TYPE XtsPartStatus :
STRUCT
	PartDriveState: Tc3_XTS_Utility.DriveState;
	IsDCLinkReady: BOOL;
	IsPartActive: BOOL;
	PartLength: LREAL;
	AllModuleSsInOP: BOOL;
END_STRUCT
END_TYPE

(* stored: Version 1.1.0.1
   DUT XtsPartStatus: Id {f04fb26b-0918-45b6-8a01-9856f31f58d4} *)
